FUNCTION_BLOCK AX_T_FF_SR_SEQ (* Event-driven bistable and Toggle, zusaetzlich echt bidirektional kettenfaehig ueber ASR2 (CHAIN_IN/CHAIN_OUT) fuer gestaffeltes Ein-/Ausschalten mehrerer Baender - Vorwaerts (CHAIN_IN.EO_SET/EO_RESET -> CHAIN_OUT.EO_SET/EO_RESET) UND Rueckwaerts (CHAIN_OUT.EI_SET/EI_RESET -> CHAIN_IN.EI_SET/EI_RESET), 4 strikt getrennte Pfade, keine Verzweigung. *)
  (* Standard: 61499-1 Annex A; Function: Lokales S/R/CLK verhaelt sich exakt wie AX_T_FF_SR und loest NIE CHAIN_IN/CHAIN_OUT aus. 4 strikt getrennte, nicht verzweigende Pfade: (1) CHAIN_IN.EO_SET -> lokal SET + CHAIN_OUT.EO_SET (Vorwaerts-Set). (2) CHAIN_IN.EO_RESET -> lokal RESET + CHAIN_OUT.EO_RESET (Vorwaerts-Reset). (3) CHAIN_OUT.EI_SET -> lokal SET + CHAIN_IN.EI_SET (Rueckwaerts-Set). (4) CHAIN_OUT.EI_RESET -> lokal RESET + CHAIN_IN.EI_RESET (Rueckwaerts-Reset). Ein ueber Pfad (1) ankommendes Set loest NIEMALS zusaetzlich Pfad (3)/(4) aus und umgekehrt - jeder Zustand feuert genau eine Chain-Aktion.; Description: Copyright (c) 2017 fortiss GmbH, HR Agrartechnik GmbH This program and the accompanying materials are made available under the terms of the Eclipse Public License 2.0 which is available at https://www.eclipse.org/legal/epl-2.0/ SPDX-License-Identifier: EPL-2.0 *)
  (* Version 1.1, 2026-09-17, Franz Höpfinger, HR Agrartechnik GmbH, Echte Bidirektionalitaet ergaenzt (Franz: 'Chain IN SET --> Chain Out Set, und Rueckwaerts auch so. keine Events verdoppeln... insgesamt 4 Pfade. keine Verzweigungen'): 2 neue Zustaende SET_CHAIN_BWD/RESET_CHAIN_BWD fuer die Rueckwaerts-Richtung (CHAIN_OUT.EI_SET/EI_RESET -> lokal + CHAIN_IN.EI_SET/EI_RESET), symmetrisch zu SET_CHAIN/RESET_CHAIN aber mit eigener, getrennter ECAction (nie CHAIN_OUT.EO_*, nur CHAIN_IN.EI_* ) - dadurch koennen z.B. Igel/Elevator/Querband ueber denselben physischen Kettenaufbau sowohl vorwaerts (SET, Downstream zuerst) als auch rueckwaerts (RESET, Upstream zuerst) gestaffelt geschaltet werden, ohne dass ein Vorwaerts-Event versehentlich auch rueckwaerts weiterlaeuft oder umgekehrt. *)
  (* Version 1.0, 2026-09-17, Franz Höpfinger, HR Agrartechnik GmbH, Kopiert von AX_T_FF_SR und um CHAIN_IN/CHAIN_OUT (ASR2-Adapter) fuer gestaffeltes kaskadiertes Set/Reset via ASR2_DELAY erweitert - lokales S/R/CLK loest CHAIN_OUT nie aus *)
  (* Version 3.0, 2025-04-14, Patrick Aigner, changed package *)
  (* Version 1.1, 2024-08-27, Franz Höpfinger, HR Agrartechnik GmbH, Copy E_SR and make this FB *)
  (* Version 1.0, 2017-09-22, Alois Zoitl, fortiss GmbH, initial API and implementation and/or initial documentation *)
  PACKAGE adapter::events::unidirectional;
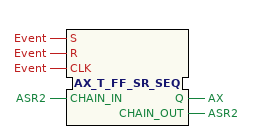
  EVENT_INPUT
    S; (* Set output Q (lokal, wirkt nie auf CHAIN_IN/CHAIN_OUT) *)
    R; (* Reset output Q (lokal, wirkt nie auf CHAIN_IN/CHAIN_OUT) *)
    CLK; (* Clock for triggering a output toggle (lokal, wirkt nie auf CHAIN_IN/CHAIN_OUT) *)
  END_EVENT
  SOCKETS
    CHAIN_IN : adapter::types::bidirectional::ASR2; (* Vorwaerts: Set/Reset vom vorherigen Kettenglied empfangen (EO_SET/EO_RESET). Rueckwaerts: Set/Reset an vorheriges Kettenglied weiterreichen (EI_SET/EI_RESET). *)
  END_SOCKETS
  PLUGS
    Q : adapter::types::unidirectional::AX; (* value of flip flop *)
    CHAIN_OUT : adapter::types::bidirectional::ASR2; (* Vorwaerts: Set/Reset an naechstes Kettenglied (EO_SET/EO_RESET). Rueckwaerts: Set/Reset VOM naechsten Kettenglied empfangen (EI_SET/EI_RESET). *)
  END_PLUGS
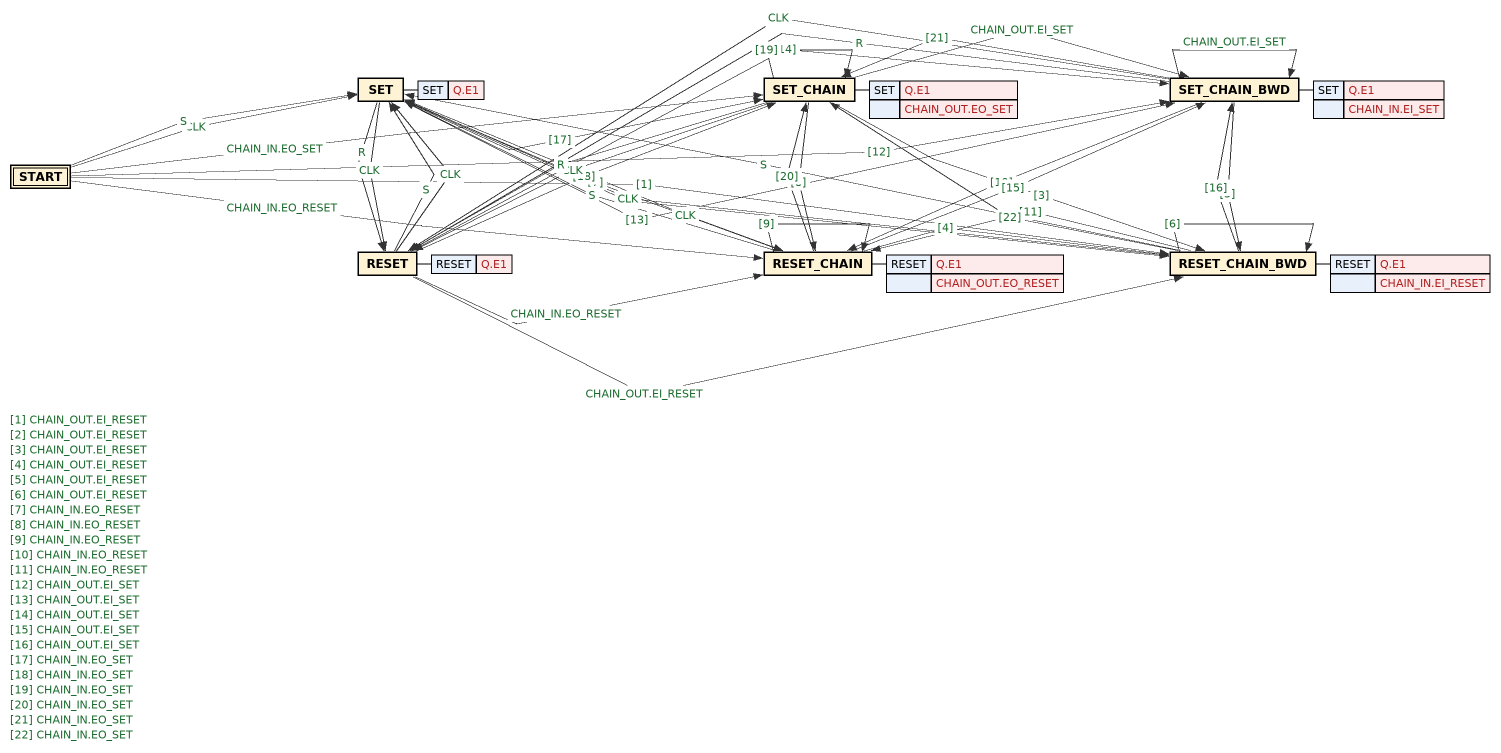
  EC_STATES
    START; (* Initial State *)
    SET : SET -> Q.E1;
    RESET : RESET -> Q.E1;
    SET_CHAIN : SET -> Q.E1, -> CHAIN_OUT.EO_SET; (* Set kam vorwaerts ueber CHAIN_IN.EO_SET - reicht NUR vorwaerts an CHAIN_OUT.EO_SET weiter *)
    RESET_CHAIN : RESET -> Q.E1, -> CHAIN_OUT.EO_RESET; (* Reset kam vorwaerts ueber CHAIN_IN.EO_RESET - reicht NUR vorwaerts an CHAIN_OUT.EO_RESET weiter *)
    SET_CHAIN_BWD : SET -> Q.E1, -> CHAIN_IN.EI_SET; (* Set kam rueckwaerts ueber CHAIN_OUT.EI_SET - reicht NUR rueckwaerts an CHAIN_IN.EI_SET weiter *)
    RESET_CHAIN_BWD : RESET -> Q.E1, -> CHAIN_IN.EI_RESET; (* Reset kam rueckwaerts ueber CHAIN_OUT.EI_RESET - reicht NUR rueckwaerts an CHAIN_IN.EI_RESET weiter *)
  END_STATES
  EC_TRANSITIONS
    START TO SET := S;
    START TO SET := CLK;
    START TO SET_CHAIN := CHAIN_IN.EO_SET;
    START TO RESET_CHAIN := CHAIN_IN.EO_RESET;
    START TO SET_CHAIN_BWD := CHAIN_OUT.EI_SET;
    START TO RESET_CHAIN_BWD := CHAIN_OUT.EI_RESET;
    SET TO RESET := R;
    SET TO RESET := CLK;
    SET TO SET_CHAIN := CHAIN_IN.EO_SET;
    SET TO RESET_CHAIN := CHAIN_IN.EO_RESET;
    SET TO SET_CHAIN_BWD := CHAIN_OUT.EI_SET;
    SET TO RESET_CHAIN_BWD := CHAIN_OUT.EI_RESET;
    RESET TO SET := S;
    RESET TO SET := CLK;
    RESET TO SET_CHAIN := CHAIN_IN.EO_SET;
    RESET TO RESET_CHAIN := CHAIN_IN.EO_RESET;
    RESET TO SET_CHAIN_BWD := CHAIN_OUT.EI_SET;
    RESET TO RESET_CHAIN_BWD := CHAIN_OUT.EI_RESET;
    SET_CHAIN TO RESET := R;
    SET_CHAIN TO RESET := CLK;
    SET_CHAIN TO SET_CHAIN := CHAIN_IN.EO_SET;
    SET_CHAIN TO RESET_CHAIN := CHAIN_IN.EO_RESET;
    SET_CHAIN TO SET_CHAIN_BWD := CHAIN_OUT.EI_SET;
    SET_CHAIN TO RESET_CHAIN_BWD := CHAIN_OUT.EI_RESET;
    RESET_CHAIN TO SET := S;
    RESET_CHAIN TO SET := CLK;
    RESET_CHAIN TO SET_CHAIN := CHAIN_IN.EO_SET;
    RESET_CHAIN TO RESET_CHAIN := CHAIN_IN.EO_RESET;
    RESET_CHAIN TO SET_CHAIN_BWD := CHAIN_OUT.EI_SET;
    RESET_CHAIN TO RESET_CHAIN_BWD := CHAIN_OUT.EI_RESET;
    SET_CHAIN_BWD TO RESET := R;
    SET_CHAIN_BWD TO RESET := CLK;
    SET_CHAIN_BWD TO SET_CHAIN := CHAIN_IN.EO_SET;
    SET_CHAIN_BWD TO RESET_CHAIN := CHAIN_IN.EO_RESET;
    SET_CHAIN_BWD TO SET_CHAIN_BWD := CHAIN_OUT.EI_SET;
    SET_CHAIN_BWD TO RESET_CHAIN_BWD := CHAIN_OUT.EI_RESET;
    RESET_CHAIN_BWD TO SET := S;
    RESET_CHAIN_BWD TO SET := CLK;
    RESET_CHAIN_BWD TO SET_CHAIN := CHAIN_IN.EO_SET;
    RESET_CHAIN_BWD TO RESET_CHAIN := CHAIN_IN.EO_RESET;
    RESET_CHAIN_BWD TO SET_CHAIN_BWD := CHAIN_OUT.EI_SET;
    RESET_CHAIN_BWD TO RESET_CHAIN_BWD := CHAIN_OUT.EI_RESET;
  END_TRANSITIONS
  ALGORITHM SET IN ST:
Q.D1 := TRUE;
  END_ALGORITHM
  ALGORITHM RESET IN ST:
Q.D1 := FALSE;
  END_ALGORITHM
END_FUNCTION_BLOCK
